// TIA Portal project "3M-8" (V16)

(* hardware
DEVICE "S7-1200 station_1"  S7-1200 Station
   slot 0: "Rack_0"  S7-1200 Rack  Rack  V1.0
   slot 1: "PLC_1"  CPU 1212C AC/DC/Rly  6ES7 212-1BE40-0XB0  V4.0
*)

// ===== PLC "PLC_1"  CPU 1212C AC/DC/Rly =====

VAR_GLOBAL   // PLC tag table "Default tag table"
   "start1" AT %I0.2 : Bool;
   "K1" AT %Q0.0 : Bool;
   "stop1" AT %I0.4 : Bool;
   "k2" AT %Q0.1 : Bool;
   "STOP" AT %I0.3 : Bool;
   "T1 tag" AT %M0.0 : Bool;
   "T2 tag" AT %M0.1 : Bool;
   "X" AT %M0.2 : Bool;
   "C1" AT %M1.0 : Bool;
   "C2" AT %M1.1 : Bool;
   "K3" AT %Q0.2 : Bool;
   "C3" AT %M1.2 : Bool;
   "C4" AT %M1.3 : Bool;
   "T3 tag" AT %M0.3 : Bool;
END_VAR

// folder: System blocks/Program resources

DATA_BLOCK "T1"   // DB2
{ S7_Optimized_Access := 'TRUE' }
AUTHOR : Simatic
FAMILY : IEC
NAME : IEC_TMR
VERSION : 1.0
// stored: InstanceOfName IEC_TIMER
"IEC_TIMER"
BEGIN
END_DATA_BLOCK

DATA_BLOCK "T2"   // DB3
{ S7_Optimized_Access := 'TRUE' }
AUTHOR : Simatic
FAMILY : IEC
NAME : IEC_TMR
VERSION : 1.0
// stored: InstanceOfName IEC_TIMER
"IEC_TIMER"
BEGIN
END_DATA_BLOCK

DATA_BLOCK "T3"   // DB4
{ S7_Optimized_Access := 'TRUE' }
AUTHOR : Simatic
FAMILY : IEC
NAME : IEC_TMR
VERSION : 1.0
// stored: InstanceOfName IEC_TIMER
"IEC_TIMER"
BEGIN
END_DATA_BLOCK

// folder: (top level)

ORGANIZATION_BLOCK "Main"   // OB1, LAD, ProgramCycle
TITLE = "Main Program Sweep (Cycle)"
{ S7_Optimized_Access := 'TRUE' }
VERSION : 0.1
   VAR_INPUT
      Initial_Call : Bool;   // Initial call of this OB
      Remanence : Bool;   // =True, if remanent data are available
   END_VAR
BEGIN

REGION Network 1: start
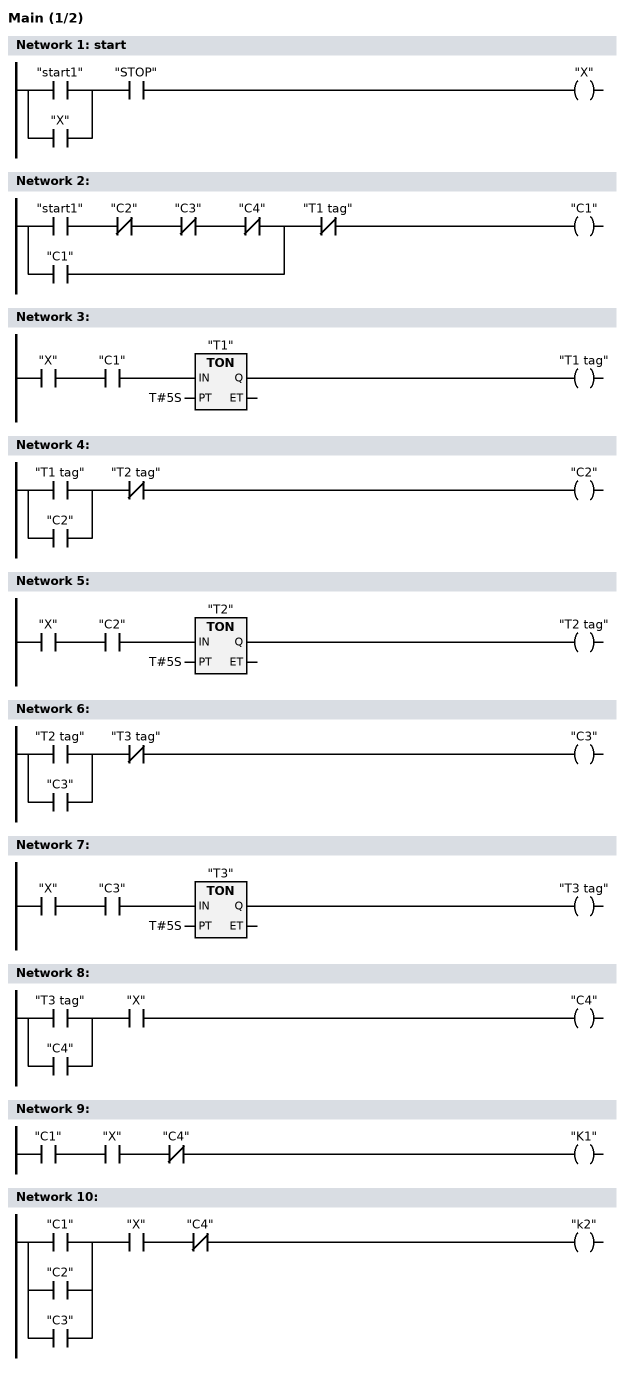
   RUNG wire#powerrail
      Contact( "start1" )
      wire#w1
      Contact( "STOP" )
      Coil( "X" )
   END_RUNG
   RUNG wire#powerrail
      Contact( "X" )
   END_RUNG wire#w1
   // the same network as SCL:
   "X" := ("start1" OR "X") AND "STOP";
END_REGION

REGION Network 2
   RUNG wire#powerrail
      Contact( "start1" )
      I_Contact( "C2" )
      I_Contact( "C3" )
      I_Contact( "C4" )
      wire#w1
      I_Contact( "T1 tag" )
      Coil( "C1" )
   END_RUNG
   RUNG wire#powerrail
      Contact( "C1" )
   END_RUNG wire#w1
   // the same network as SCL:
   "C1" := (("start1" AND NOT "C2" AND NOT "C3" AND NOT "C4") OR "C1") AND NOT "T1 tag";
END_REGION

REGION Network 3
   "T1".TON(IN := "X" AND "C1", PT := T#5S);
   "T1 tag" := "T1".Q;
END_REGION

REGION Network 4
   RUNG wire#powerrail
      Contact( "T1 tag" )
      wire#w1
      I_Contact( "T2 tag" )
      Coil( "C2" )
   END_RUNG
   RUNG wire#powerrail
      Contact( "C2" )
   END_RUNG wire#w1
   // the same network as SCL:
   "C2" := ("T1 tag" OR "C2") AND NOT "T2 tag";
END_REGION

REGION Network 5
   "T2".TON(IN := "X" AND "C2", PT := T#5S);
   "T2 tag" := "T2".Q;
END_REGION

REGION Network 6
   RUNG wire#powerrail
      Contact( "T2 tag" )
      wire#w1
      I_Contact( "T3 tag" )
      Coil( "C3" )
   END_RUNG
   RUNG wire#powerrail
      Contact( "C3" )
   END_RUNG wire#w1
   // the same network as SCL:
   "C3" := ("T2 tag" OR "C3") AND NOT "T3 tag";
END_REGION

REGION Network 7
   "T3".TON(IN := "X" AND "C3", PT := T#5S);
   "T3 tag" := "T3".Q;
END_REGION

REGION Network 8
   RUNG wire#powerrail
      Contact( "T3 tag" )
      wire#w1
      Contact( "X" )
      Coil( "C4" )
   END_RUNG
   RUNG wire#powerrail
      Contact( "C4" )
   END_RUNG wire#w1
   // the same network as SCL:
   "C4" := ("T3 tag" OR "C4") AND "X";
END_REGION

REGION Network 9
   RUNG wire#powerrail
      Contact( "C1" )
      Contact( "X" )
      I_Contact( "C4" )
      Coil( "K1" )
   END_RUNG
   // the same network as SCL:
   "K1" := "C1" AND "X" AND NOT "C4";
END_REGION

REGION Network 10
   RUNG wire#powerrail
      Contact( "C1" )
      wire#w1
      Contact( "X" )
      I_Contact( "C4" )
      Coil( "k2" )
   END_RUNG
   RUNG wire#powerrail
      Contact( "C2" )
   END_RUNG wire#w1
   RUNG wire#powerrail
      Contact( "C3" )
   END_RUNG wire#w1
   // the same network as SCL:
   "k2" := ("C1" OR "C2" OR "C3") AND "X" AND NOT "C4";
END_REGION

REGION Network 11
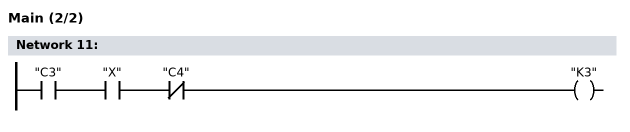
   RUNG wire#powerrail
      Contact( "C3" )
      Contact( "X" )
      I_Contact( "C4" )
      Coil( "K3" )
   END_RUNG
   // the same network as SCL:
   "K3" := "C3" AND "X" AND NOT "C4";
END_REGION
END_ORGANIZATION_BLOCK